# EPICS StreamDevice protocol: apps/dynapowerApp/Db/dynapower-2022.proto
OutTerminator = CR;
#InTerminator = LF CR;
InTerminator = ;

keepalive { out ""; }
putHex    { out "SET\$1%.2x"; }
putFloat  { out "SET\$1%.0f"; }
putString { out "SET\$1%s"; }

# The documentation came with getters but they do not work,
# instead the strings below are sent every 2 seconds.
#getHex    { out "GET \$1"; in "%x"; }
#getFloat  { out "GET \$1"; in "%f"; }

# Have seen all of these with a bit different terminations:
# \r\n 1 \r\n 7 \r\n 712 \r\n 0 \r\n 0010 \r\n 0000 \r\n 0000\r\n07\036\r\000\000\000\000\000\000\000\000\000\000\000\000
# \r\n 1 \r\n 7 \r\n 712 \r\n 0 \r\n 0010 \r\n 0000 \r\n 0000\r\n\n\r\036\r\000\000\000\000\000\000\000\000\000\000\000\000
# \r\n 1 \r\n 7 \r\n 712 \r\n 0 \r\n 0010 \r\n 0000 \r\n 0000\r\n0\r\036\r\000\000\000\000\000\000\000\000\000\000\000\000

# Also seen this, with values that do not look physical, and much different termination:
# \r\n 1 \r\n 7 \r\n 1356 \r\n 500 \r\n 0010 \r\n 0000 \r\n 0000\r\036\r\000\000\000\000\000\000\000\000\000\000\000\000

# Catch the first three, ignore the other one:
getVolt { extrainput=ignore; in " \r\n %d \r\n %*d \r\n %*d \r\n %*d \r\n %*x \r\n %*x \r\n %*x\r\n"; }
getAmps { extrainput=ignore; in " \r\n %*d \r\n %d \r\n %*d \r\n %*d \r\n %*x \r\n %*x \r\n %*x\r\n"; }
getTemp { extrainput=ignore; in " \r\n %*d \r\n %*d \r\n %d \r\n %*d \r\n %*x \r\n %*x \r\n %*x\r\n"; }
getFlow { extrainput=ignore; in " \r\n %*d \r\n %*d \r\n %*d \r\n %d \r\n %*x \r\n %*x \r\n %*x\r\n"; }
getStat { extrainput=ignore; in " \r\n %*d \r\n %*d \r\n %*d \r\n %*d \r\n %x \r\n %*x \r\n %*x\r\n"; }
getFlt1 { extrainput=ignore; in " \r\n %*d \r\n %*d \r\n %*d \r\n %*d \r\n %*x \r\n %x \r\n %*x\r\n"; }
getFlt2 { extrainput=ignore; in " \r\n %*d \r\n %*d \r\n %*d \r\n %*d \r\n %*x \r\n %*x \r\n %x\r\n"; }
